FUNCTION F_Replace : STRING(255)
VAR_INPUT
	sInputText		:STRING(255);
	sSearchText		:STRING(255);
	sReplaceText	:STRING(255);
END_VAR
VAR
	idxFnd			:INT;
	iLength			:INT;
END_VAR

idxFnd := FIND(sInputText, sSearchText);
iLength := LEN(sSearchText);

IF idxFnd > 0 THEN
	F_Replace := REPLACE(sInputText, sReplaceText, iLength, idxFnd);
ELSE
	F_Replace := sInputText;
END_IF

END_FUNCTION

(* stored: Version 1.1.0.1, ProductVersion 3.1.4024.11
   POU F_Replace: Id {bc2cd2d9-5a7c-4421-8368-d99a6888382b}, SpecialFunc None *)
